# EPICS StreamDevice protocol: protocols/hudp.proto
Terminator = LF;
ExtraInput = Ignore;

getIp {
	out "ip";
	in "%s";
}

getDstIp {
	out "dst_ip";
	in "%s";
}

getDstPort {
	out "dst_port";
	in "%d";
}

getTxPktSz {
	out "tx_calc_pkt_sz";
	in "%d";
}

getTxSPP {
	out "tx_spp";
	in "%d";
}

getRxSrcIp {
	out "rx_src_ip";
	in "%s";
}

getRxPort {
	out "rx_port";
	in "%d";
}

getRxPktLen {
	out "rx_pkt_len";
	in "%d";
}

setCtrlEnum {
	out "tx_ctrl %{0|9|1}";
	in "";
}

getCtrlEnum {
	out "ctrl";
	in "%{0|9|1}";
}

getCtrlRaw {
	out "ctrl";
	in "%d";
}

setCtrlRaw {
	out "ctrl %d";
	in "";
}

getDiscoEn {
	out "disco_en";
	in "%d";
}

setDiscoEn {
	out "disco_en %d";
	in "";
}

getDiscoIdx {
	out "disco_idx";
	in "%d";
}

setDiscoIdx {
	out "disco_idx %d";
	in "";
}

setUdpDataSrc {
	out "udp_data_src %d";
	in "";
}
